
FUNCTION FC23 : VOID
//QBLOCK
Author:'RJ'
VAR_INPUT
    IN:REAL;
END_VAR

VAR_OUTPUT
    OUT:REAL;
END_VAR
    OUT:=IN;
END_FUNCTION
